// TIA Portal V20 export
DATA_BLOCK "EeMonitorData"   // DB108
TITLE = EeMonitorData
AUTHOR : SICAR
FAMILY : DB
// Energy efficency monitor Daten / Energy efficency monitor data
// stored: InstanceOfName LSicar_typeEemData, InstanceOfType UDT
"LSicar_typeEemData"
   // VAR
   //    machineConfiguration : EnS_EEm_typeConfig;
   //    machineOperation : EnS_EEm_typeOperation;
   //    measConfiguration : Array[0..9] of EnS_EEm_typeMeasConfig;
   //    measOperation : Array[0..9] of EnS_EEm_typeMeasOperation;
   //    internalData : "LSicar_typeEemDataInternal";
   //    calcError : Bool := FALSE;
   //    calcStatus : Word := 16#740B;
   //    calcRetVal : Int := 0;
   //    reportCreateCsv : Bool := FALSE;
   //    reportStatus : Word := 16#0000;
   //    reportNameCsv : String[80] := '';
   // END_VAR
BEGIN
   machineConfiguration."name" := 'Default_Machine_Demo';
   machineConfiguration."type" := 'Default_Type_Demo';
   machineConfiguration.serialNumber := 'Default_Serial_Number_Demo';
   machineConfiguration.manufacturer := 'Default_Manufacturer_Demo';
   machineConfiguration.licenseKey := 'Demo_Demo_Demo_Demo!';
   machineConfiguration.pieceOverflowCntValue := 10000.0;
   machineConfiguration.eStateName[0] := 'Undefined';
   machineConfiguration.eStateName[1] := 'Auto';
   machineConfiguration.eStateName[2] := 'Auto Preselect';
   machineConfiguration.eStateName[3] := 'Manual';
   machineConfiguration.eStateName[4] := 'Idle';
   machineConfiguration.eStateName[5] := 'Fault';
   machineConfiguration.eStateName[6..8] := '-Not used-';
   machineConfiguration.additionalInfoDescription[0] := 'additional Info1';
   machineConfiguration.additionalInfoDescription[1] := 'additional Info2';
   machineConfiguration.additionalInfoDescription[2] := 'additional Info3';
   machineConfiguration.additionalInfoDescription[3] := 'additional Info4';
   machineOperation.pieceCounter := 0.0;
   machineOperation.additionalInformation[0] := 'AddInfo 1';
   machineOperation.additionalInformation[1] := 'AddInfo 2';
   machineOperation.additionalInformation[2] := 'AddInfo 3';
   machineOperation.additionalInformation[3] := 'AddInfo 4';
   machineOperation.eState := 0;
   machineOperation.maskEnPI := 16#0002;
   machineOperation.triggerRecalcOutput := FALSE;
   machineOperation.resetMeasErrors := FALSE;
   machineOperation.globalResetEnergyCounter := FALSE;
   machineOperation.globalResetAvgValues := FALSE;
   machineOperation.globalResetEnergyPerItem := FALSE;
   machineOperation.startAvgCalcPeriod := FALSE;
   machineOperation.stopAvgCalcPeriod := FALSE;
   machineOperation.setAvgCalcRef := FALSE;
   machineOperation.stat.arraysOk := TRUE;
   machineOperation.stat.avgCalcAct := FALSE;
   machineOperation.stat.triggerRecalcOld := FALSE;
   machineOperation.stat.startAvgCalcOld := FALSE;
   machineOperation.stat.stopAvgCalcOld := FALSE;
   machineOperation.stat.referenceAvgCalcSave := FALSE;
   machineOperation.stat.outputValuesRelease := TRUE;
   machineOperation.stat.maskEnpiOld := 16#0002;
   machineOperation.stat.machineEStateOld := 0;
   machineOperation.stat.upBoundMeasConfiguration := 9;
   machineOperation.stat.upBoundMeasOperation := 9;
   machineOperation.stat.lowBoundMeasConfiguration := 0;
   machineOperation.stat.lowBoundMeasOperation := 0;
   machineOperation.stat.pieceCntOld := 0.0;
   machineOperation.stat.pieceCntEnpiCalc := 0.0;
   machineOperation.stat.cycleCounterAvgCalc := 0;
   machineOperation.stat.cycleCounterEstates[0..8] := 0;
   machineOperation.stat.startTimeAvgVal := DTL#1970-01-01-00:00:00;
   machineOperation.stat.timePeriodAvgVal := T#0MS;
   machineOperation.stat.timeZoneValues := T#0MS;
   machineOperation.stat.startTimeAvgRef := DTL#1970-01-01-00:00:00;
   machineOperation.stat.timePeriodAvgRef := T#0MS;
   machineOperation.stat.timeZoneRef := T#0MS;
   machineOperation.stat.systemInformation[0] := 16#07;
   machineOperation.stat.systemInformation[1] := 16#EA;
   machineOperation.stat.systemInformation[2] := 16#01;
   machineOperation.stat.systemInformation[3] := 16#06;
   machineOperation.stat.systemInformation[4] := 16#03;
   machineOperation.stat.systemInformation[5] := 16#05;
   machineOperation.stat.systemInformation[6] := 16#09;
   machineOperation.stat.systemInformation[7] := 16#2B;
   machineOperation.stat.systemInformation[8] := 16#03;
   machineOperation.stat.systemInformation[9] := 16#CC;
   machineOperation.stat.systemInformation[10] := 16#19;
   machineOperation.stat.systemInformation[11] := 16#C5;
   measConfiguration[0]."name" := 'AIEnergyMeter480VACST_EM01';
   measConfiguration[1]."name" := 'AIEnergyMeter480VACST_EM02';
   measConfiguration[2]."name" := 'PAC Electrical Infeed';
   measConfiguration[3..9]."name" := 'MeasPointXX';
   measConfiguration[0].nameShort := 'EM01';
   measConfiguration[1].nameShort := 'EM02';
   measConfiguration[2].nameShort := 'P01';
   measConfiguration[3..9].nameShort := 'XX01';
   measConfiguration[0..9].media := 'electrical';
   measConfiguration[0..9].unitCounterNumber := 1;
   measConfiguration[0..9].unitCounterText := 'Wh';
   measConfiguration[0..9].unitActValueNumber := 0;
   measConfiguration[0..9].unitActValueText := 'W';
   measConfiguration[0..9].inputType := 1;
   measConfiguration[0..9].type1Counter.overflowCntValue := 1000000.0;
   measConfiguration[0..9].type1Counter.normFactor := 1.0;
   measConfiguration[0..9].type2ActValue.rawLow := 0.0;
   measConfiguration[0..9].type2ActValue.rawHigh := 100.0;
   measConfiguration[0..9].type2ActValue.outLow := 0.0;
   measConfiguration[0..9].type2ActValue.outHigh := 100.0;
   measOperation[0].in.counterValue := 277.384918212891;
   measOperation[1..9].in.counterValue := 0.0;
   measOperation[0..9].in.actValue := 0.0;
   measOperation[0].out.avgValue[0..8] := 0.0;
   measOperation[1].out.avgValue[0..8] := 0.0;
   measOperation[2].out.avgValue[0..8] := 0.0;
   measOperation[3].out.avgValue[0..8] := 0.0;
   measOperation[4].out.avgValue[0..8] := 0.0;
   measOperation[5].out.avgValue[0..8] := 0.0;
   measOperation[6].out.avgValue[0..8] := 0.0;
   measOperation[7].out.avgValue[0..8] := 0.0;
   measOperation[8].out.avgValue[0..8] := 0.0;
   measOperation[9].out.avgValue[0..8] := 0.0;
   measOperation[0].out.refValue[0..8] := 0.0;
   measOperation[1].out.refValue[0..8] := 0.0;
   measOperation[2].out.refValue[0..8] := 0.0;
   measOperation[3].out.refValue[0..8] := 0.0;
   measOperation[4].out.refValue[0..8] := 0.0;
   measOperation[5].out.refValue[0..8] := 0.0;
   measOperation[6].out.refValue[0..8] := 0.0;
   measOperation[7].out.refValue[0..8] := 0.0;
   measOperation[8].out.refValue[0..8] := 0.0;
   measOperation[9].out.refValue[0..8] := 0.0;
   measOperation[0].out.differencePercent[0..8] := 0.0;
   measOperation[1].out.differencePercent[0..8] := 0.0;
   measOperation[2].out.differencePercent[0..8] := 0.0;
   measOperation[3].out.differencePercent[0..8] := 0.0;
   measOperation[4].out.differencePercent[0..8] := 0.0;
   measOperation[5].out.differencePercent[0..8] := 0.0;
   measOperation[6].out.differencePercent[0..8] := 0.0;
   measOperation[7].out.differencePercent[0..8] := 0.0;
   measOperation[8].out.differencePercent[0..8] := 0.0;
   measOperation[9].out.differencePercent[0..8] := 0.0;
   measOperation[0].out.energyCounter[0] := 4.5557861328125;
   measOperation[0].out.energyCounter[1..8] := 0.0;
   measOperation[1].out.energyCounter[0..8] := 0.0;
   measOperation[2].out.energyCounter[0..8] := 0.0;
   measOperation[3].out.energyCounter[0..8] := 0.0;
   measOperation[4].out.energyCounter[0..8] := 0.0;
   measOperation[5].out.energyCounter[0..8] := 0.0;
   measOperation[6].out.energyCounter[0..8] := 0.0;
   measOperation[7].out.energyCounter[0..8] := 0.0;
   measOperation[8].out.energyCounter[0..8] := 0.0;
   measOperation[9].out.energyCounter[0..8] := 0.0;
   measOperation[0].out.energyCounterTotal := 4.5557861328125;
   measOperation[1..9].out.energyCounterTotal := 0.0;
   measOperation[0..9].out.error := FALSE;
   measOperation[0..9].out.energyPerItem := 0.0;
   measOperation[0].stat.counterLast := 277.473693847656;
   measOperation[1..9].stat.counterLast := 0.0;
   measOperation[0].stat.counterDifference := 277.384918212891;
   measOperation[1..9].stat.counterDifference := 0.0;
   measOperation[0].stat.startEnergyValue[0..8] := 0.0;
   measOperation[1].stat.startEnergyValue[0..8] := 0.0;
   measOperation[2].stat.startEnergyValue[0..8] := 0.0;
   measOperation[3].stat.startEnergyValue[0..8] := 0.0;
   measOperation[4].stat.startEnergyValue[0..8] := 0.0;
   measOperation[5].stat.startEnergyValue[0..8] := 0.0;
   measOperation[6].stat.startEnergyValue[0..8] := 0.0;
   measOperation[7].stat.startEnergyValue[0..8] := 0.0;
   measOperation[8].stat.startEnergyValue[0..8] := 0.0;
   measOperation[9].stat.startEnergyValue[0..8] := 0.0;
   measOperation[0..9].stat.energyCounterIntermediate := 0.0;
   measOperation[0].stat.energyEnPiCalc[0] := 4.555786;
   measOperation[0].stat.energyEnPiCalc[1..8] := 0.0;
   measOperation[1].stat.energyEnPiCalc[0..8] := 0.0;
   measOperation[2].stat.energyEnPiCalc[0..8] := 0.0;
   measOperation[3].stat.energyEnPiCalc[0..8] := 0.0;
   measOperation[4].stat.energyEnPiCalc[0..8] := 0.0;
   measOperation[5].stat.energyEnPiCalc[0..8] := 0.0;
   measOperation[6].stat.energyEnPiCalc[0..8] := 0.0;
   measOperation[7].stat.energyEnPiCalc[0..8] := 0.0;
   measOperation[8].stat.energyEnPiCalc[0..8] := 0.0;
   measOperation[9].stat.energyEnPiCalc[0..8] := 0.0;
   internalData.productiveEnergyStates[0] := FALSE;
   internalData.productiveEnergyStates[1] := TRUE;
   internalData.productiveEnergyStates[2..8] := FALSE;
   internalData.enpiGoals[0..9] := 0.0;
   internalData.enpiResetTrigger := FALSE;
   internalData.enpiResetTime := DTL#1970-01-01-00:00:00;
   internalData.measPointConfiguration.measPointName := '';
   internalData.measPointConfiguration.measPointMedia := '';
   internalData.measPointConfiguration.measPointUnitCounter := '';
   internalData.measPointConfiguration.measPointUnitActual := '';
   internalData.measPointConfiguration.measPointType := 0;
   internalData.measPointConfiguration.measPointType1Overflow := 0.0;
   internalData.measPointConfiguration.measPointType1NormFactor := 0.0;
   internalData.measPointConfiguration.measPointType2RawLow := 0.0;
   internalData.measPointConfiguration.measPointType2RawHigh := 0.0;
   internalData.measPointConfiguration.measPointType2OutLow := 0.0;
   internalData.measPointConfiguration.measPointType2OutHigh := 0.0;
   internalData.measPointConfiguration.measPointDataSave := FALSE;
   internalData.measPointConfiguration.measPointDataRead := FALSE;
   internalData.measPointConfiguration.measPointInitializationCancel := FALSE;
   internalData.measPointConfiguration.measPointDataWritten := 0;
   internalData.measPointConfiguration.measPointDataIndex := 0;
   internalData.measPointConfiguration.numberMeasPoints := 0;
   internalData.measPointConfiguration.measPointInitialized := FALSE;
   internalData.enmProEnabled := FALSE;
   internalData.enmProData.state := 16#0000;
   internalData.enmProData.error := FALSE;
   internalData.enmProData.save := FALSE;
   internalData.enmProData.abort := FALSE;
   internalData.enmProData.ipAdress[1..4] := 0;
   internalData.enmProData.localPort := 3000;
   internalData.enmProData.remotePort := 3000;
   internalData.enmProData.interfaceId := 64;
   internalData.enmProData.connectionId := 16#000E;
END_DATA_BLOCK
